Omron CX-Programmer project NuevoProyecto (CX-Programmer 9.81)

# PLC NuevoPLC1: CJ1M CPU11

## Global symbols (name address type ; comment)
0.00 BOOL  ; encendido
10.00 BOOL  ; verde
10.01 BOOL  ; AMARILLO
10.02 BOOL  ; ROJA

## Program NuevoPrograma1 (cyclic task 0)

### Section Sección1

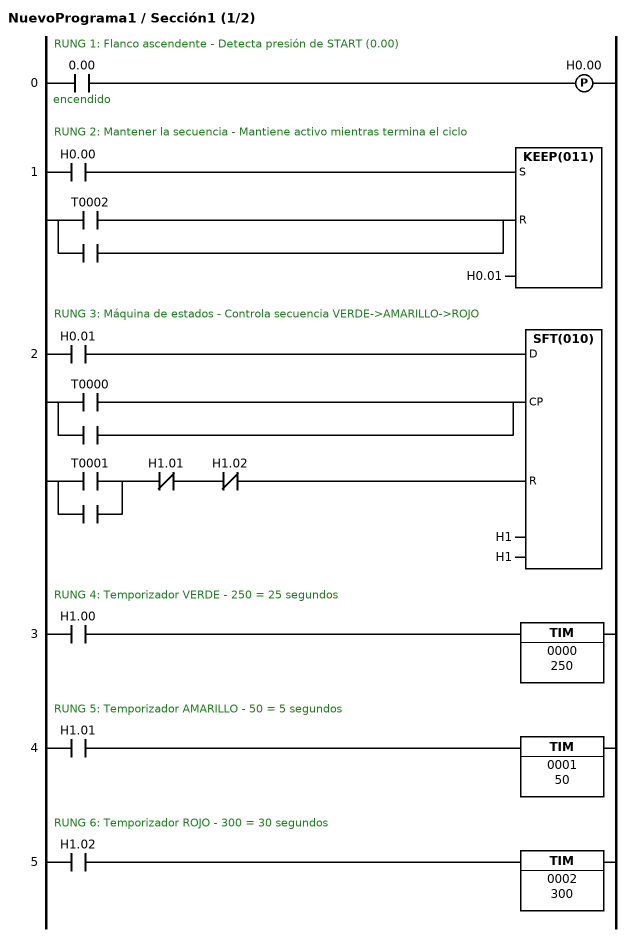
; rung 0: RUNG 1: Flanco ascendente - Detecta presión de START (0.00)
LD 0.00  ; encendido
DIFU(013) H0.00
; rung 1: RUNG 2: Mantener la secuencia - Mantiene activo mientras termina el ciclo
LD H0.00
LD T0002
OR
KEEP(011) H0.01
; rung 2: RUNG 3: Máquina de estados - Controla secuencia VERDE->AMARILLO->ROJO
LD H0.01
LD T0000
OR
LD T0001
OR
ANDNOT H1.01
ANDNOT H1.02
SFT(010) H1 H1
; rung 3: RUNG 4: Temporizador VERDE - 250 = 25 segundos
LD H1.00
TIM 0000 250
; rung 4: RUNG 5: Temporizador AMARILLO - 50 = 5 segundos
LD H1.01
TIM 0001 50
; rung 5: RUNG 6: Temporizador ROJO - 300 = 30 segundos
LD H1.02
TIM 0002 300

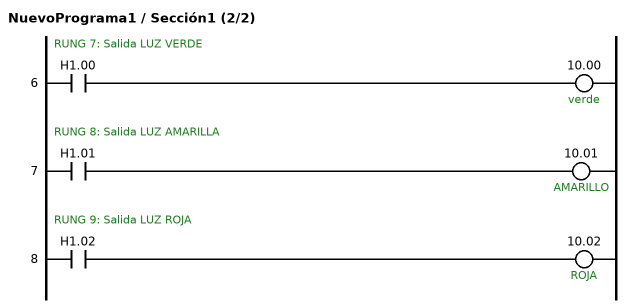
; rung 6: RUNG 7: Salida LUZ VERDE
LD H1.00
OUT 10.00  ; verde
; rung 7: RUNG 8: Salida LUZ AMARILLA
LD H1.01
OUT 10.01  ; AMARILLO
; rung 8: RUNG 9: Salida LUZ ROJA
LD H1.02
OUT 10.02  ; ROJA

### Section END
; rung 0
END(001)